{attribute 'qualified_only'}
{attribute 'strict'}
TYPE DigitalInputStatus:
(
        LOW := 0,
        HIGH := 1
);
END_TYPE

(* stored: Version 1.1.0.1, ProductVersion 3.1.4024.12
   DUT DigitalInputStatus: Id {d7c1a315-09b7-423e-96dc-15fca2f70cd8} *)
